// TIA Portal project "Lab03-modbus" (V16)

(* hardware
DEVICE "S7-1200 station_1"  S7-1200 Station
   slot 0: "Rack_0"  S7-1200 Rack  Rack  V1.0
   slot 1: "PLC_1"  CPU 1212C DC/DC/DC  6ES7 212-1AE40-0XB0  V4.4
*)

// ===== PLC "PLC_1"  CPU 1212C DC/DC/DC =====

VAR_GLOBAL   // PLC tag table "Tabla de variables estándar"
   "Clock_Byte" AT %MB0 : Byte;
   "Clock_10Hz" AT %M0.0 : Bool;
   "Clock_5Hz" AT %M0.1 : Bool;
   "Clock_2.5Hz" AT %M0.2 : Bool;
   "Clock_2Hz" AT %M0.3 : Bool;
   "Clock_1.25Hz" AT %M0.4 : Bool;
   "Clock_1Hz" AT %M0.5 : Bool;
   "Clock_0.625Hz" AT %M0.6 : Bool;
   "Clock_0.5Hz" AT %M0.7 : Bool;
   "System_Byte" AT %MB1 : Byte;
   "FirstScan" AT %M1.0 : Bool;
   "DiagStatusUpdate" AT %M1.1 : Bool;
   "AlwaysTRUE" AT %M1.2 : Bool;
   "AlwaysFALSE" AT %M1.3 : Bool;
   "AUX1" AT %M2.0 : Bool;
END_VAR

DATA_BLOCK "MB_Server_Connect"   // DB1
{ S7_Optimized_Access := 'TRUE' }
VERSION : 0.1
   VAR
      Connect : TCON_IP_v4;
   END_VAR
BEGIN
   Connect.InterfaceId := 64;
   Connect.ID := 1;
   Connect.ConnectionType := 11;
   Connect.RemoteAddress.ADDR[1] := 192;
   Connect.RemoteAddress.ADDR[2] := 168;
   Connect.RemoteAddress.ADDR[3] := 0;
   Connect.RemoteAddress.ADDR[4] := 20;
   Connect.LocalPort := 502;
END_DATA_BLOCK

DATA_BLOCK "MB_Holding_Register"   // DB2
{ S7_Optimized_Access := 'FALSE' }
VERSION : 0.1
   VAR
      HR1 : Int;
      HR2 : Int;
      HR3 : Int;
      HR4 : Int;
      HR5 : Int;
      HR6 : Int;
      HR7 : Int;
      HR8 : Int;
      HR9 : Int;
      HR10 : Int;
   END_VAR
BEGIN
END_DATA_BLOCK

FUNCTION "FC_MB_Server" : Void   // FC1, LAD
{ S7_Optimized_Access := 'TRUE' }
VERSION : 0.1
   VAR_TEMP   // added for the SCL form of the ladder/FBD networks
      _w1 : Bool;
   END_VAR
BEGIN

REGION Network 1
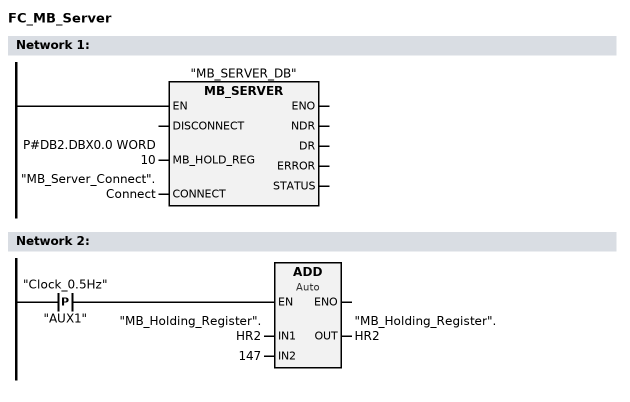
   "MB_SERVER_DB"(MB_HOLD_REG := P#DB2.DBX0.0 WORD 10, CONNECT := "MB_Server_Connect".Connect);   // MB_SERVER
END_REGION

REGION Network 2
   RUNG wire#powerrail
      P_Contact(operand := "Clock_0.5Hz", bit := "AUX1")
      Add(in1 := "MB_Holding_Register".HR2, in2 := 147, out => "MB_Holding_Register".HR2)
   END_RUNG
   // the same network as SCL:
   #_w1 := "Clock_0.5Hz" AND NOT "AUX1";   // rising edge of "Clock_0.5Hz"
   "AUX1" := "Clock_0.5Hz";
   IF #_w1 THEN "MB_Holding_Register".HR2 := "MB_Holding_Register".HR2 + 147; END_IF;
END_REGION
END_FUNCTION

ORGANIZATION_BLOCK "Main"   // OB1, LAD, ProgramCycle
TITLE = "Main Program Sweep (Cycle)"
{ S7_Optimized_Access := 'TRUE' }
VERSION : 0.1
   VAR_INPUT
      Initial_Call : Bool;   // Initial call of this OB
      Remanence : Bool;   // =True, if remanent data are available
   END_VAR
BEGIN

REGION Network 1
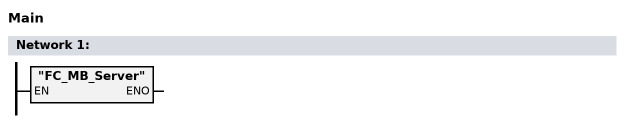
   RUNG wire#powerrail
      "FC_MB_Server"()
   END_RUNG
   // the same network as SCL:
   "FC_MB_Server"();
END_REGION
END_ORGANIZATION_BLOCK